(* PLC project TimerTest *)
(* stored: creationDateTime 2024-01-01T00:00:00, modificationDateTime 2024-01-01T00:00:00 *)

PROGRAM Main
  VAR
    X001 : BOOL;
    T001 : BOOL;
    Y001 : BOOL;
    T001_Instance : TON;
  END_VAR

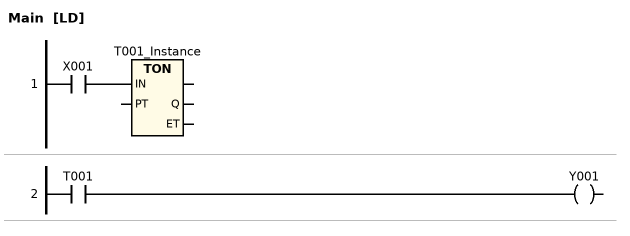
(* LD diagram, written out as Structured Text *)
Y001 := T001;
T001_Instance(IN := X001);
END_PROGRAM

CONFIGURATION Config
  RESOURCE Res ON PLC
    TASK Main(INTERVAL := T#20ms, PRIORITY := 0);
    PROGRAM Main WITH Main : Main;
  END_RESOURCE
END_CONFIGURATION
